// TIA Portal V20 export
DATA_BLOCK "DB_HmiKeyboardSignals"   // DB90
// stored: InstanceOfName FB_HmiKeyboardSignals, InstanceOfType FB
"FB_HmiKeyboardSignals"
   // VAR
   //    sK1_Powermeter : "FB_HmiKeysSignalsManu";
   //    sK2_GasAssist { S7_SetPoint := 'True'} : "FB_HmiKeysSignalsManu";
   //    sK4a_GripperUndrilledPartClose { S7_SetPoint := 'True'} : "FB_HmiKeysSignalsManu";
   //    sK4b_GripperUndrilledPartOpen { S7_SetPoint := 'True'} : "FB_HmiKeysSignalsManu";
   //    sK5a_GripperDrilledPartClose { S7_SetPoint := 'True'} : "FB_HmiKeysSignalsManu";
   //    sK5b_GripperDrilledPartOpen { S7_SetPoint := 'True'} : "FB_HmiKeysSignalsManu";
   //    sK6_SITestStop { S7_SetPoint := 'True'} : "FB_HmiKeysSignalsManu";
   //    sK7_FixtureClamp { S7_SetPoint := 'True'} : "FB_HmiKeysSignalsManu";
   //    sK8_FixtureVacuum { S7_SetPoint := 'True'} : "FB_HmiKeysSignalsManu";
   //    sK9_Aspiration { S7_SetPoint := 'True'} : "FB_HmiKeysSignalsManu";
   //    sK12a_Backlight { S7_SetPoint := 'True'} : "FB_HmiKeysSignalsManu";
   //    sK12b_ObservationCamera { S7_SetPoint := 'True'} : "FB_HmiKeysSignalsManu";
   //    sK13_MainDoor { S7_SetPoint := 'True'} : "FB_HmiKeysSignalsManu";
   //    sK14_WarmUp { S7_SetPoint := 'True'} : "FB_HmiKeysSignalsManu";
   //    sK15_MachineLight { S7_SetPoint := 'True'} : "FB_HmiKeysSignalsManu";
   // END_VAR
BEGIN
END_DATA_BLOCK
